FUNCTION_BLOCK Scale (* Basic Function Block Type *)
  (* Standard: 61499-2 *)
  (* Version 0.0, 24/05/2016, Chen-Wei, nxtControl GmbH, Template *)
  PACKAGE Main;
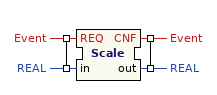
  EVENT_INPUT
    REQ WITH in; (* Normal Execution Request *)
  END_EVENT
  EVENT_OUTPUT
    CNF WITH out; (* Execution Confirmation *)
  END_EVENT
  VAR_INPUT
    in : REAL; (* Input event qualifier *)
  END_VAR
  VAR_OUTPUT
    out : REAL; (* Output event qualifier *)
  END_VAR
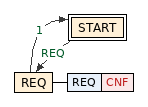
  EC_STATES
    START; (* Initial State *)
    REQ : REQ -> CNF; (* Normal execution *)
  END_STATES
  EC_TRANSITIONS
    START TO REQ := REQ;
    REQ TO START := 1;
  END_TRANSITIONS
  ALGORITHM INIT IN ST: (* Initialization algorithm *)
;
  END_ALGORITHM
  ALGORITHM REQ IN ST: (* Normally executed algorithm *)
REQ := 0;

out := in/10;

;
  END_ALGORITHM
END_FUNCTION_BLOCK
